TYPE ST_FileExtensions :
STRUCT
	Text	: STRING := '.txt';
	Csv		: STRING := '.csv';
END_STRUCT
END_TYPE

(* stored: Version 1.1.0.1, ProductVersion 3.1.4024.13
   DUT ST_FileExtensions: Id {d30f35df-a5fa-0d23-05d3-b6da271b8347} *)
